TYPE StepAction :
STRUCT
	name			: STRING;
	number			: INT;
	description		: STRING;
	timeout			: TIME;
END_STRUCT
END_TYPE

(* stored: Version 1.1.0.1, ProductVersion 3.1.4024.11
   DUT StepAction: Id {0b353818-406c-4514-93dc-ab01f8b8d470} *)
